Fanuc KAREL source: kb00077.KL

-- PROVISIONAL review KL for V770-1; original PC SHA256 e33138cffa0be0e71a6b3a5b9e1e6ce0129514b23deec27e327ee17308e0e4c4
-- Incomplete behavior may be omitted. Consult companion uncertainty JSON. Do not deploy.
PROGRAM KB00077
%NOLOCKGROUP
BEGIN
  -- UNRESOLVED_PC offsets 5-14; opcodes 3F,75
  -- UNRESOLVED_PC offsets 19-26; opcodes 9D,23
  -- UNRESOLVED_PC offsets 31-38; opcodes 9D,23
  -- UNRESOLVED_PC offsets 43-52; opcodes 3F,75
  -- UNRESOLVED_PC offsets 57-64; opcodes 9D,23
  -- UNRESOLVED_PC offsets 69-107; opcodes 27,22,2A,22,22,22,2A,22,31
  -- UNRESOLVED_PC offsets 112-116; opcodes 7F
END KB00077
